(* IEC 61131-3 sources: repolevel_ST_code_completion/real_groud_truth最新/repoeval_traffic_light/full_result, 3 files *)

(* ---- F_SecondsToTime.st ---- *)
FUNCTION F_SecondsToTime : TIME
VAR_INPUT
	dwSeconds	:	DWORD;		//输入的秒数
END_VAR

// 将秒数（DWORD）转换为TIME类型
    // TIME类型内部是以毫秒为单位存储的，因此需要将秒数乘以1000
    F_SecondsToTime := DWORD_TO_TIME(dwSeconds * 1000);
END_FUNCTION

(* ---- F_TimeToSeconds.st ---- *)
FUNCTION F_TimeToSeconds : DWORD
VAR_INPUT
	tTime	:	TIME;		//输入的时间
END_VAR

// 将TIME类型转换为秒数（DWORD）
    F_TimeToSeconds := TIME_TO_DWORD(tTime) / 1000;
END_FUNCTION

(* ---- FB_CountdownTimer.st ---- *)
FUNCTION_BLOCK FB_CountdownTimer
VAR_INPUT
	tElapsedTime	:	TIME;		//已经过的时间（定时器的ET）
	tTotalTime		:	TIME;		//总时间（定时器的PT）
END_VAR
VAR_OUTPUT
	nRemainingSeconds	:	UINT;	//剩余秒数
END_VAR

VAR
	tRemainingTime	:	TIME;		//剩余时间
END_VAR

// 计算剩余时间
tRemainingTime := tTotalTime - tElapsedTime;

// 如果剩余时间小于零，则设置为零
IF tRemainingTime < T#0ms THEN
	tRemainingTime := T#0ms;
END_IF

// 将剩余时间转换为秒数
nRemainingSeconds := TIME_TO_UINT(TRUNC(TIME_TO_DWORD(tRemainingTime) / 1000.0));
END_FUNCTION_BLOCK
